INTERFACE ITF_1_Communication

METHOD Connect : BOOL
VAR_INPUT
END_VAR
END_METHOD

PROPERTY Connected : BOOL
GET
END_GET
END_PROPERTY

METHOD Disconnect : BOOL
VAR_INPUT
END_VAR
END_METHOD

METHOD Reconnect : BOOL
VAR_INPUT
END_VAR
END_METHOD

METHOD Send : BOOL
VAR_INPUT
      pData : PVOID;
      nDataSize : UDINT;
END_VAR
END_METHOD

METHOD Update : BOOL
VAR_INPUT
END_VAR
END_METHOD

END_INTERFACE

(* stored: Version 1.1.0.1, ProductVersion 3.1.4026.18
   Itf ITF_1_Communication: Id {137062f4-e0da-4742-8af0-d297ced283f8}
   Method Connect: Id {87cfa5c5-c74d-443b-add2-3a7c89de83c3}
   Property Connected: Id {e3a4778a-0f53-4054-bb5d-4b61ee314b7b}
   Get Get: Id {c9e26e2d-8e27-47d9-95e7-96b913ca6803}
   Method Disconnect: Id {c9f14a31-d44b-4480-9761-6c4eb27b28db}
   Method Reconnect: Id {bf377ed8-2360-417f-9da3-0098c69dbfd2}
   Method Send: Id {fbb76a85-3e04-4d63-ace1-c87edd3b98a3}
   Method Update: Id {1e26b47d-130f-40af-81c4-fb80dc20112f} *)
